ABB RobotStudio station: Basics1.rspag

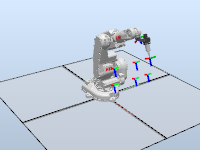
--- station ---
Station Basics1 (saved by RobotStudio 21.2.9526.0)
Controller CRB1100_4_47_Controller
  mechanical unit ROB_1: IRB140_6_81_C_03, 6 joints, base frame (0, 0, 0) mm
Layout (positions relative to the parent item):
  - IRB140_6_81_C_03 [mechanism, from Robots\IRB140_6_81_C_G_03.rslib] at (0, 0, 0) mm; joint values [0.0303, 0.1039, -0.5495, -0.0318, 0.9697, 0.0331] (rad or m)
  - MyTool [mechanism, from Training Objects\myTool.rslib] at (506.29, 13.63, 841.36) mm, rotated rx 180 ry 60 rz 180 deg
Attachment: MyTool is attached to IRB140_6_81_C_03 / Link6
Targets, tools, work objects and paths stored in the station and not in the controller backup, written as RAPID:
! task T_ROB1
MODULE CalibData
  PERS tooldata MyTool:=[TRUE,[[31.792631019,0,229.638935148],[0.945518576,0,0.325568154,0]],[1,[0,0,1],[1,0,0,0],0,0,0]];
ENDMODULE

! task T_ROB1
MODULE Module1
  CONST robtarget Target_10:=[[689.268561308,0,537.147252465],[0.190808931,0,0.981627196,0],[0,0,0,0],[9E+09,9E+09,9E+09,9E+09,9E+09,9E+09]];
  CONST robtarget Target_20:=[[689.268622176,-149.172609109,537.147198426],[0.190808859,0.000000009,0.98162721,0.000000003],[-1,0,-1,0],[9E+09,9E+09,9E+09,9E+09,9E+09,9E+09]];
  CONST robtarget Target_40:=[[689.268626986,-387.821682782,537.14720904],[0.190808863,-0.000000011,0.981627209,0.000000002],[-1,0,-1,0],[9E+09,9E+09,9E+09,9E+09,9E+09,9E+09]];
  CONST robtarget Target_60:=[[689.268613221,-387.821697865,699.010297051],[0.190808762,0.000000001,0.981627229,0.000000022],[-1,0,-1,0],[9E+09,9E+09,9E+09,9E+09,9E+09,9E+09]];
  CONST robtarget Target_80:=[[689.268623901,-150.604388741,699.010277632],[0.190808752,0.00000001,0.981627231,0.000000024],[-1,0,-1,0],[9E+09,9E+09,9E+09,9E+09,9E+09,9E+09]];
  CONST robtarget Target_100:=[[689.268613687,13.631250255,699.010282713],[0.190808743,0.000000009,0.981627233,0.000000024],[0,-1,0,0],[9E+09,9E+09,9E+09,9E+09,9E+09,9E+09]];
ENDMODULE


--- Backups/CRB1100_4_47_Controller/RAPID/TASK1/PROGMOD/Module1.mod ---
MODULE Module1
    !***********************************************************
    !
    ! Module:  Module1
    !
    ! Description:
    !   <Insert description here>
    !
    ! Author: mateusz
    !
    ! Version: 1.0
    !
    !***********************************************************


    !***********************************************************
    !
    ! Procedure main
    !
    !   This is the entry point of your program
    !
    !***********************************************************
    PROC main()
        !Add your code here
    ENDPROC
ENDMODULE
